// Mitsubishi GX Works2 project: JOG 제어, 원점 복귀, 위치 결정 데이터 복합 코드   PLC: Q03UDV

PROGRAM MAIN
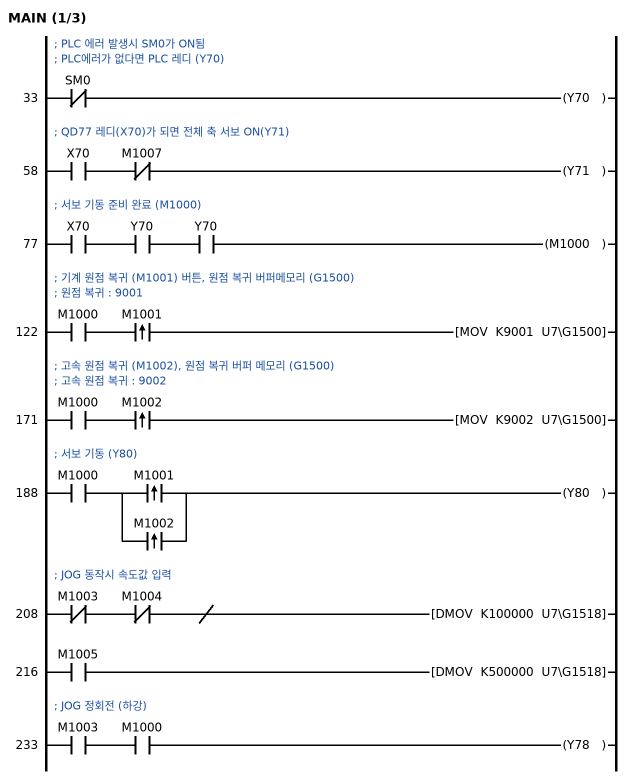
; PLC 에러 발생시 SM0가 ON됨
; PLC에러가 없다면 PLC 레디 (Y70)
33    LDI     SM0
      OUT     Y70
; QD77 레디(X70)가 되면 전체 축 서보 ON(Y71)
58    LD      X70
      ANI     M1007
      OUT     Y71
; 서보 기동 준비 완료 (M1000)
77    LD      X70
      AND     Y70
      AND     Y70
      OUT     M1000
; 기계 원점 복귀 (M1001) 버튼, 원점 복귀 버퍼메모리 (G1500)
; 원점 복귀 : 9001
122   LD      M1000
      ANDP    M1001
      MOV     K9001 U7\G1500
; 고속 원점 복귀 (M1002), 원점 복귀 버퍼 메모리 (G1500)
; 고속 원점 복귀 : 9002
171   LD      M1000
      ANDP    M1002
      MOV     K9002 U7\G1500
; 서보 기동 (Y80)
188   LD      M1000
      LDP     M1001
      ORP     M1002
      ANB
      OUT     Y80
; JOG 동작시 속도값 입력
208   LDI     M1003
      ANI     M1004
      INV
      DMOV    K100000 U7\G1518
216   LD      M1005
      DMOV    K500000 U7\G1518
; JOG 정회전 (하강)
233   LD      M1003
      AND     M1000
      OUT     Y78
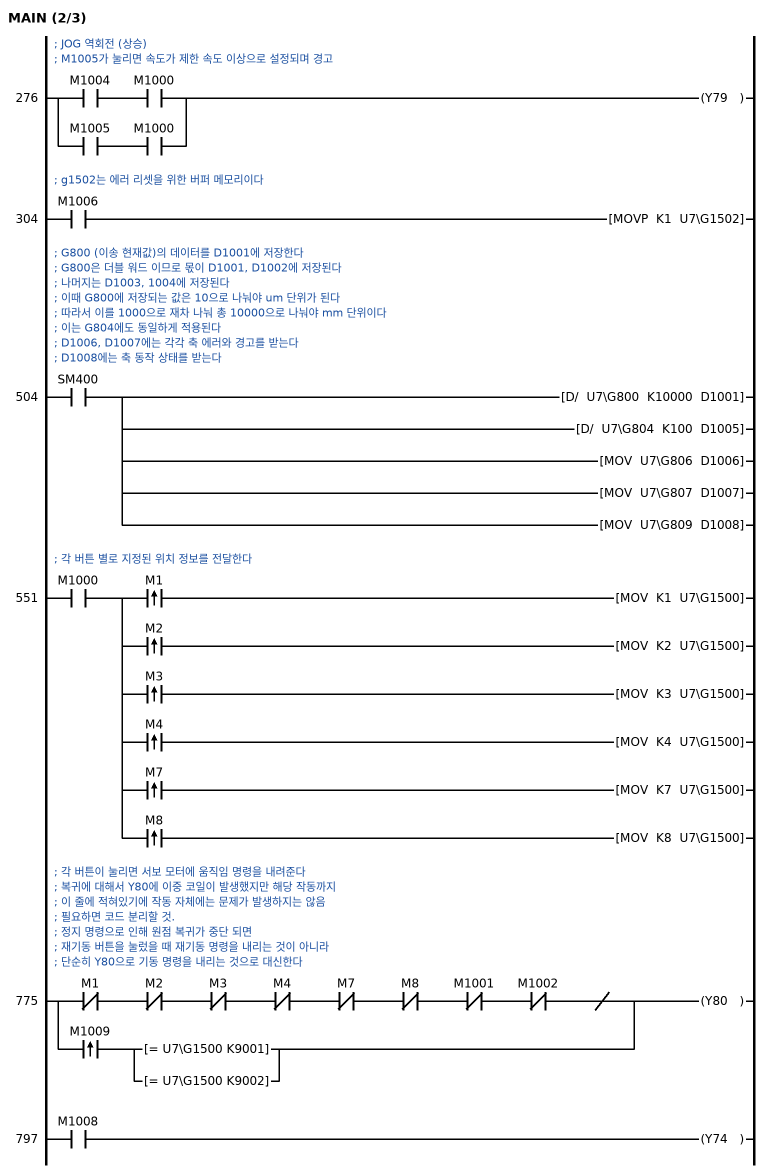
; JOG 역회전 (상승)
; M1005가 눌리면 속도가 제한 속도 이상으로 설정되며 경고
276   LD      M1004
      AND     M1000
      LD      M1005
      AND     M1000
      ORB
      OUT     Y79
; g1502는 에러 리셋을 위한 버퍼 메모리이다
304   LD      M1006
      MOVP    K1 U7\G1502
; G800 (이송 현재값)의 데이터를 D1001에 저장한다
; G800은 더블 워드 이므로 몫이 D1001, D1002에 저장된다
; 나머지는 D1003, 1004에 저장된다
; 이때 G800에 저장되는 값은 10으로 나눠야 um 단위가 된다
; 따라서 이를 1000으로 재차 나눠 총 10000으로 나눠야 mm 단위이다
; 이는 G804에도 동일하게 적용된다
; D1006, D1007에는 각각 축 에러와 경고를 받는다
; D1008에는 축 동작 상태를 받는다
504   LD      SM400
      D/      U7\G800 K10000 D1001
      D/      U7\G804 K100 D1005
      MOV     U7\G806 D1006
      MOV     U7\G807 D1007
      MOV     U7\G809 D1008
; 각 버튼 별로 지정된 위치 정보를 전달한다
551   LD      M1000
      MPS
      ANDP    M1
      MOV     K1 U7\G1500
      MRD
      ANDP    M2
      MOV     K2 U7\G1500
      MRD
      ANDP    M3
      MOV     K3 U7\G1500
      MRD
      ANDP    M4
      MOV     K4 U7\G1500
      MRD
      ANDP    M7
      MOV     K7 U7\G1500
      MPP
      ANDP    M8
      MOV     K8 U7\G1500
; 각 버튼이 눌리면 서보 모터에 움직임 명령을 내려준다
; 복귀에 대해서 Y80에 이중 코일이 발생했지만 해당 작동까지
; 이 줄에 적혀있기에 작동 자체에는 문제가 발생하지는 않음
; 필요하면 코드 분리할 것.
; 정지 명령으로 인해 원점 복귀가 중단 되면
; 재기동 버튼을 눌렀을 때 재기동 명령을 내리는 것이 아니라
; 단순히 Y80으로 기동 명령을 내리는 것으로 대신한다
775   LDI     M1
      ANI     M2
      ANI     M3
      ANI     M4
      ANI     M7
      ANI     M8
      ANI     M1001
      ANI     M1002
      INV
      LDP     M1009
      LD=     U7\G1500 K9001
      OR=     U7\G1500 K9002
      ANB
      ORB
      OUT     Y80
797   LD      M1008
      OUT     Y74
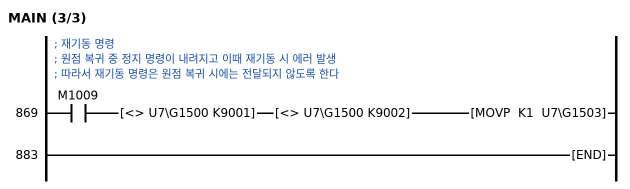
; 재기동 명령
; 원점 복귀 중 정지 명령이 내려지고 이때 재기동 시 에러 발생
; 따라서 재기동 명령은 원점 복귀 시에는 전달되지 않도록 한다
869   LD      M1009
      AND<>   U7\G1500 K9001
      AND<>   U7\G1500 K9002
      MOVP    K1 U7\G1503
883   END
END_PROGRAM
